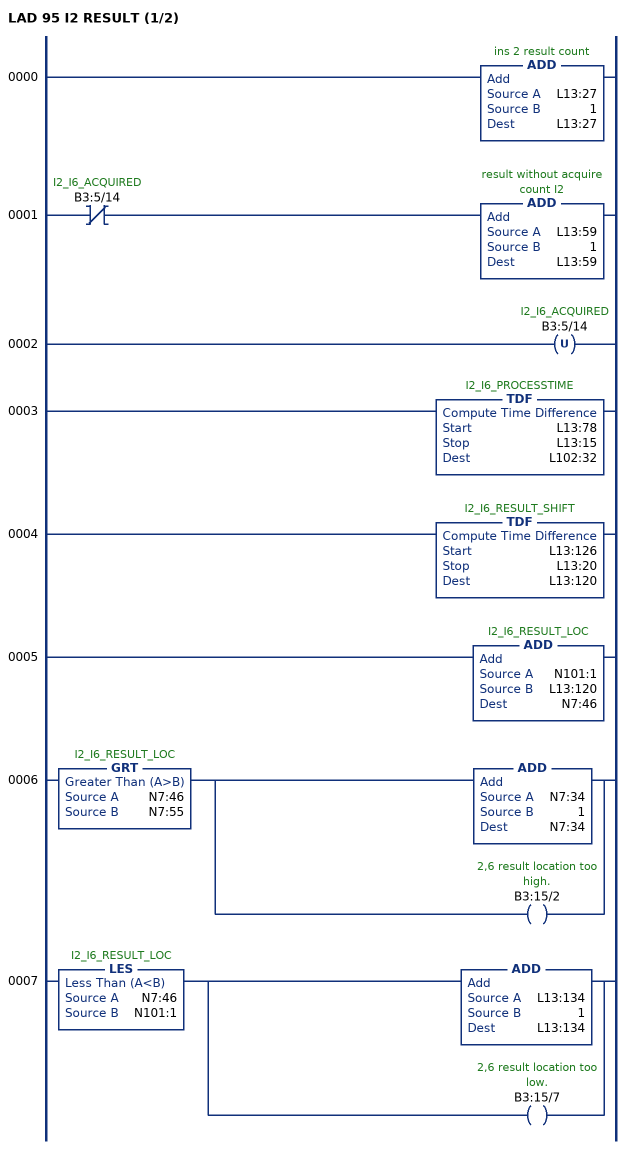
% Rung: 0 %
SOR ADD L13:27 1 L13:27 EOR
%   L13:27  "ins 2 result count" %
% Rung: 1 %
SOR XIO B3:5/14 ADD L13:59 1 L13:59 EOR
%   B3:5/14  I2_I6_ACQUIRED %
%   L13:59  "result without acquire count I2" %
% Rung: 2 %
SOR OTU B3:5/14 EOR
%   B3:5/14  I2_I6_ACQUIRED %
% Rung: 3 %
SOR TDF L13:78 L13:15 L102:32 EOR
%   L13:78  I2_I6_TIMEOFACQ %
%   L13:15  THE_TIME %
%   L102:32  I2_I6_PROCESSTIME %
% Rung: 4 %
SOR TDF L13:126 L13:20 L13:120 EOR
%   L13:126  I2_I6_PROC_START_POS %
%   L13:20  BOT_POSITION %
%   L13:120  I2_I6_RESULT_SHIFT %
% Rung: 5 %
SOR ADD N101:1 L13:120 N7:46 EOR
%   N101:1  I2_TRIG_LOC %
%   L13:120  I2_I6_RESULT_SHIFT %
%   N7:46  I2_I6_RESULT_LOC %
% Rung: 6 %
SOR GRT N7:46 N7:55 BST ADD N7:34 1 N7:34 NXB OTE B3:15/2 BND EOR
%   N7:46  I2_I6_RESULT_LOC %
%   N7:55  I2_MAX_SHIFT %
%   B3:15/2  "2,6 result location too high." %
% Rung: 7 %
SOR LES N7:46 N101:1 BST ADD L13:134 1 L13:134 NXB OTE B3:15/7 BND EOR
%   N7:46  I2_I6_RESULT_LOC %
%   N101:1  I2_TRIG_LOC %
%   B3:15/7  "2,6 result location too low." %

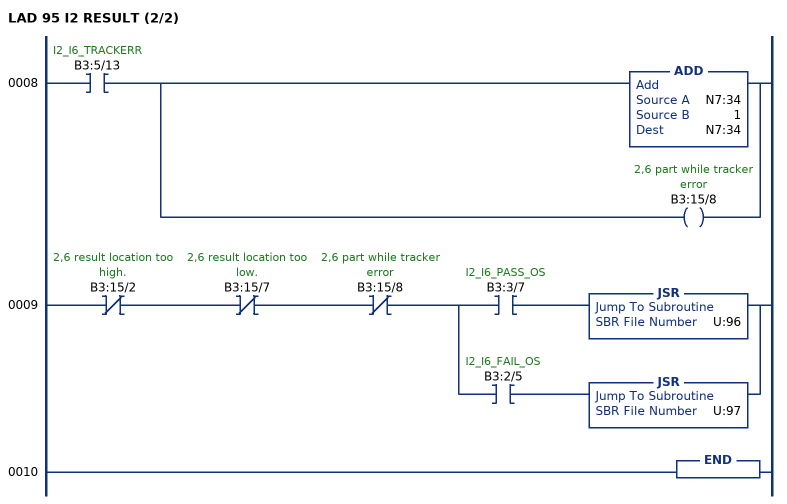
% Rung: 8 %
SOR XIC B3:5/13 BST ADD N7:34 1 N7:34 NXB OTE B3:15/8 BND EOR
%   B3:5/13  I2_I6_TRACKERR %
%   B3:15/8  "2,6 part while tracker error" %
% Rung: 9 %
SOR XIO B3:15/2 XIO B3:15/7 XIO B3:15/8 BST XIC B3:3/7 JSR U:96 NXB XIC B3:2/5 JSR U:97 BND EOR
%   B3:15/2  "2,6 result location too high." %
%   B3:15/7  "2,6 result location too low." %
%   B3:15/8  "2,6 part while tracker error" %
%   B3:3/7  I2_I6_PASS_OS %
%   B3:2/5  I2_I6_FAIL_OS %
% Rung: 10 %
SOR END EOR

LADDER 96 "I2 PASS"
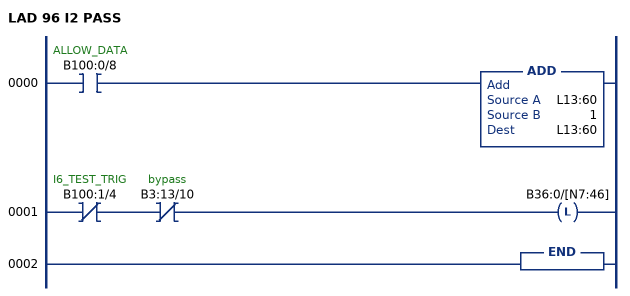
% Rung: 0 %
SOR XIC B100:0/8 ADD L13:60 1 L13:60 EOR
%   B100:0/8  ALLOW_DATA %
% Rung: 1 %
SOR XIO B100:1/4 XIO B3:13/10 OTL B36:0/[N7:46] EOR
%   B100:1/4  I6_TEST_TRIG %
%   B3:13/10  "bypass" %
%   B36:0  BOT_OK %
%   N7:46  I2_I6_RESULT_LOC %
% Rung: 2 %
SOR END EOR

LADDER 97 "I2 FAIL"
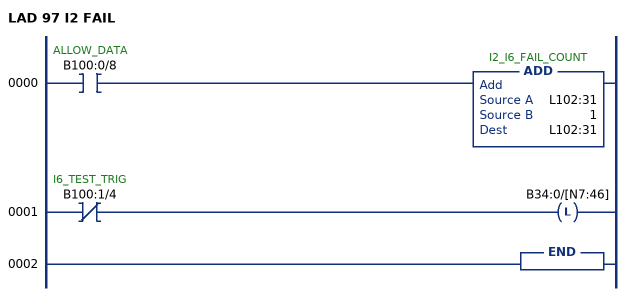
% Rung: 0 %
SOR XIC B100:0/8 ADD L102:31 1 L102:31 EOR
%   B100:0/8  ALLOW_DATA %
%   L102:31  I2_I6_FAIL_COUNT %
% Rung: 1 %
SOR XIO B100:1/4 OTL B34:0/[N7:46] EOR
%   B100:1/4  I6_TEST_TRIG %
%   B34:0  BOT_NG %
%   N7:46  I2_I6_RESULT_LOC %
% Rung: 2 %
SOR END EOR

LADDER 98 "I2 ACQ"
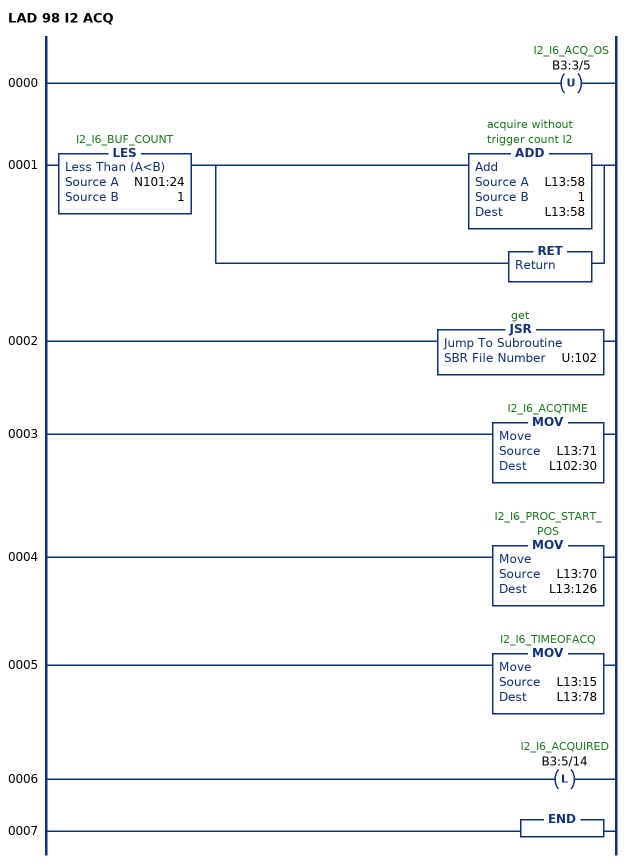
% Rung: 0 %
SOR OTU B3:3/5 EOR
%   B3:3/5  I2_I6_ACQ_OS %
% Rung: 1 %
SOR LES N101:24 1 BST ADD L13:58 1 L13:58 NXB RET BND EOR
%   N101:24  I2_I6_BUF_COUNT %
%   L13:58  "acquire without trigger count I2" %
% Rung: 2 %
SOR JSR U:102 EOR
%   U:102  "get" %
% Rung: 3 %
SOR MOV L13:71 L102:30 EOR
%   L13:71  I2_I6_TIME_SPAN %
%   L102:30  I2_I6_ACQTIME %
% Rung: 4 %
SOR MOV L13:70 L13:126 EOR
%   L13:70  I2_I6_PULLED_POS %
%   L13:126  I2_I6_PROC_START_POS %
% Rung: 5 %
SOR MOV L13:15 L13:78 EOR
%   L13:15  THE_TIME %
%   L13:78  I2_I6_TIMEOFACQ %
% Rung: 6 %
SOR OTL B3:5/14 EOR
%   B3:5/14  I2_I6_ACQUIRED %
% Rung: 7 %
SOR END EOR

LADDER 99 "I2 TESTER"
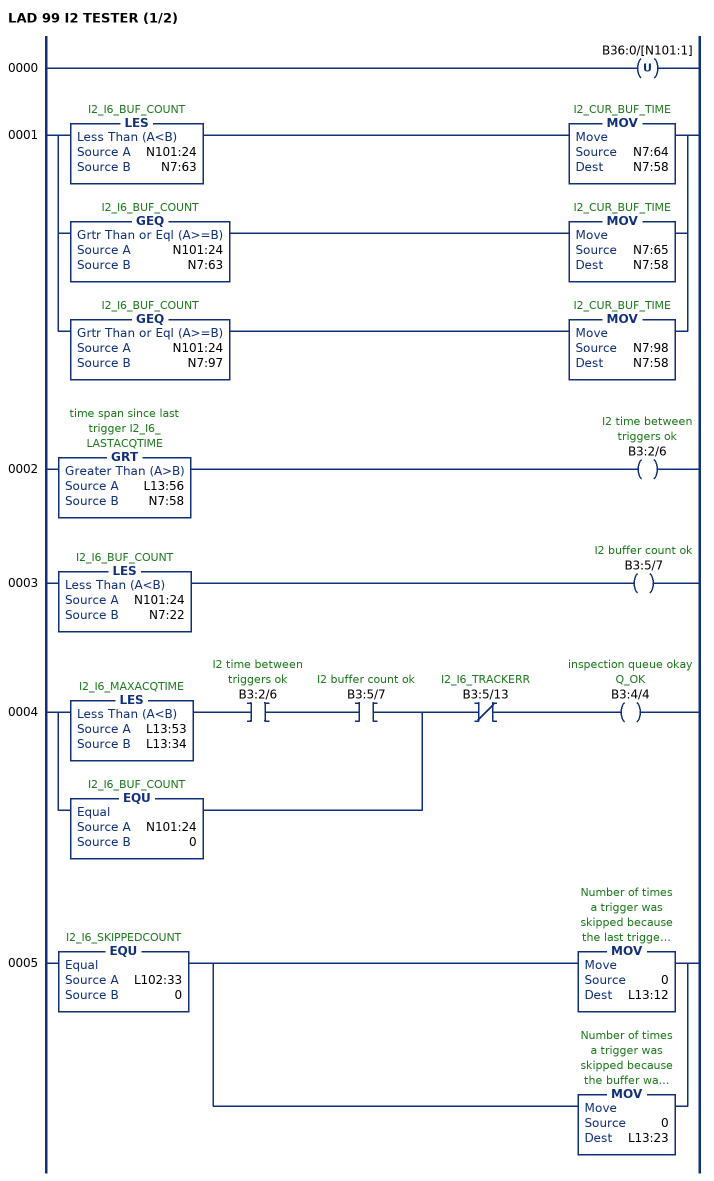
% Rung: 0 %
SOR OTU B36:0/[N101:1] EOR
%   B36:0  BOT_OK %
%   N101:1  I2_TRIG_LOC %
% Rung: 1 %
SOR BST LES N101:24 N7:63 MOV N7:64 N7:58 NXB GEQ N101:24 N7:63 MOV N7:65 N7:58 NXB GEQ N101:24 N7:97 MOV N7:98 N7:58 BND EOR
%   N101:24  I2_I6_BUF_COUNT %
%   N7:64  I2_CAM_BUF_TIME %
%   N7:58  I2_CUR_BUF_TIME %
%   N7:65  I2_PC_BUF_TIME %
% Rung: 2 %
SOR GRT L13:56 N7:58 OTE B3:2/6 EOR
%   L13:56  I2_I6_LASTACQTIME  "time span since last trigger" %
%   N7:58  I2_CUR_BUF_TIME %
%   B3:2/6  "I2 time between triggers ok" %
% Rung: 3 %
SOR LES N101:24 N7:22 OTE B3:5/7 EOR
%   N101:24  I2_I6_BUF_COUNT %
%   N7:22  MAX_BUF_ALL  "max buffer count alowed before bypass" %
%   B3:5/7  "I2 buffer count ok" %
% Rung: 4 %
SOR BST LES L13:53 L13:34 XIC B3:2/6 XIC B3:5/7 NXB EQU N101:24 0 BND XIO B3:5/13 OTE B3:4/4 EOR
%   L13:53  I2_I6_MAXACQTIME %
%   L13:34  MAX_ACQ_ALL  "absolute max acquire time before bypass trigger" %
%   B3:2/6  "I2 time between triggers ok" %
%   B3:5/7  "I2 buffer count ok" %
%   N101:24  I2_I6_BUF_COUNT %
%   B3:5/13  I2_I6_TRACKERR %
%   B3:4/4  Q_OK  "inspection queue okay" %
% Rung: 5 %
SOR EQU L102:33 0 BST MOV 0 L13:12 NXB MOV 0 L13:23 BND EOR
%   L102:33  I2_I6_SKIPPEDCOUNT %
%   L13:12  I2_FAST_TRIG_COUNT  "Number of times a trigger was skipped because the last trigger was too recent." %
%   L13:23  I2_BUF_FILL_COUNT  "Number of times a trigger was skipped because the buffer was full." %

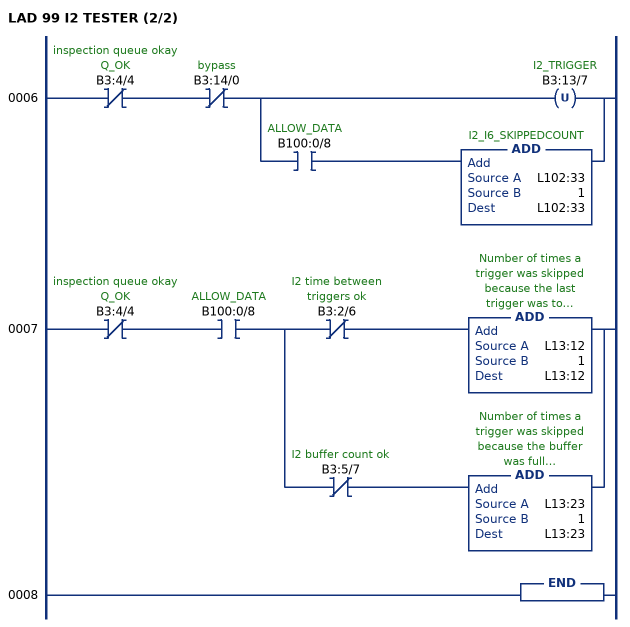
% Rung: 6 %
SOR XIO B3:4/4 XIO B3:14/0 BST OTU B3:13/7 NXB XIC B100:0/8 ADD L102:33 1 L102:33 BND EOR
%   B3:4/4  Q_OK  "inspection queue okay" %
%   B3:14/0  "bypass" %
%   B3:13/7  I2_TRIGGER %
%   B100:0/8  ALLOW_DATA %
%   L102:33  I2_I6_SKIPPEDCOUNT %
% Rung: 7 %
SOR XIO B3:4/4 XIC B100:0/8 BST XIO B3:2/6 ADD L13:12 1 L13:12 NXB XIO B3:5/7 ADD L13:23 1 L13:23 BND EOR
%   B3:4/4  Q_OK  "inspection queue okay" %
%   B100:0/8  ALLOW_DATA %
%   B3:2/6  "I2 time between triggers ok" %
%   L13:12  I2_FAST_TRIG_COUNT  "Number of times a trigger was skipped because the last trigger was too recent." %
%   B3:5/7  "I2 buffer count ok" %
%   L13:23  I2_BUF_FILL_COUNT  "Number of times a trigger was skipped because the buffer was full." %
% Rung: 8 %
SOR END EOR

LADDER 100 "I2 TRIG"
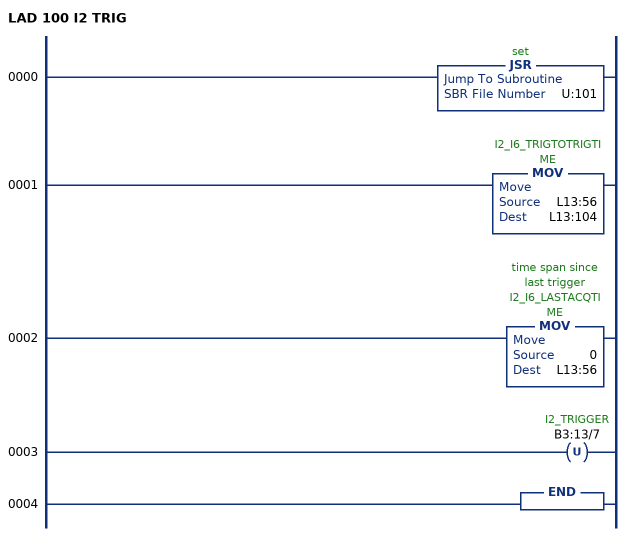
% Rung: 0 %
SOR JSR U:101 EOR
%   U:101  "set" %
% Rung: 1 %
SOR MOV L13:56 L13:104 EOR
%   L13:56  I2_I6_LASTACQTIME  "time span since last trigger" %
%   L13:104  I2_I6_TRIGTOTRIGTIME %
% Rung: 2 %
SOR MOV 0 L13:56 EOR
%   L13:56  I2_I6_LASTACQTIME  "time span since last trigger" %
% Rung: 3 %
SOR OTU B3:13/7 EOR
%   B3:13/7  I2_TRIGGER %
% Rung: 4 %
SOR END EOR

LADDER 101 "I2 FIFOSET"
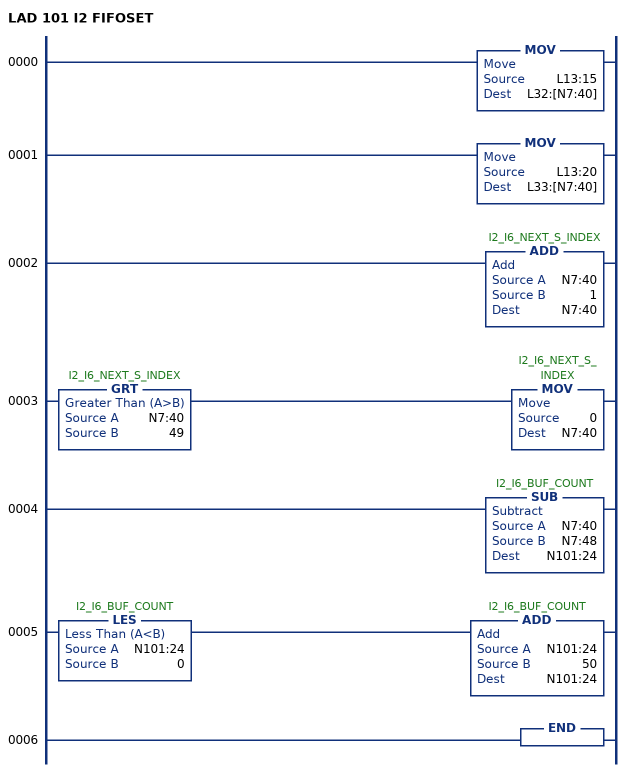
% Rung: 0 %
SOR MOV L13:15 L32:[N7:40] EOR
%   L13:15  THE_TIME %
%   N7:40  I2_I6_NEXT_S_INDEX %
% Rung: 1 %
SOR MOV L13:20 L33:[N7:40] EOR
%   L13:20  BOT_POSITION %
%   N7:40  I2_I6_NEXT_S_INDEX %
% Rung: 2 %
SOR ADD N7:40 1 N7:40 EOR
%   N7:40  I2_I6_NEXT_S_INDEX %
% Rung: 3 %
SOR GRT N7:40 49 MOV 0 N7:40 EOR
%   N7:40  I2_I6_NEXT_S_INDEX %
% Rung: 4 %
SOR SUB N7:40 N7:48 N101:24 EOR
%   N7:40  I2_I6_NEXT_S_INDEX %
%   N7:48  I2_I6_NEXT_G_INDEX %
%   N101:24  I2_I6_BUF_COUNT %
% Rung: 5 %
SOR LES N101:24 0 ADD N101:24 50 N101:24 EOR
%   N101:24  I2_I6_BUF_COUNT %
% Rung: 6 %
SOR END EOR

LADDER 102 "I2 FIFOGET"
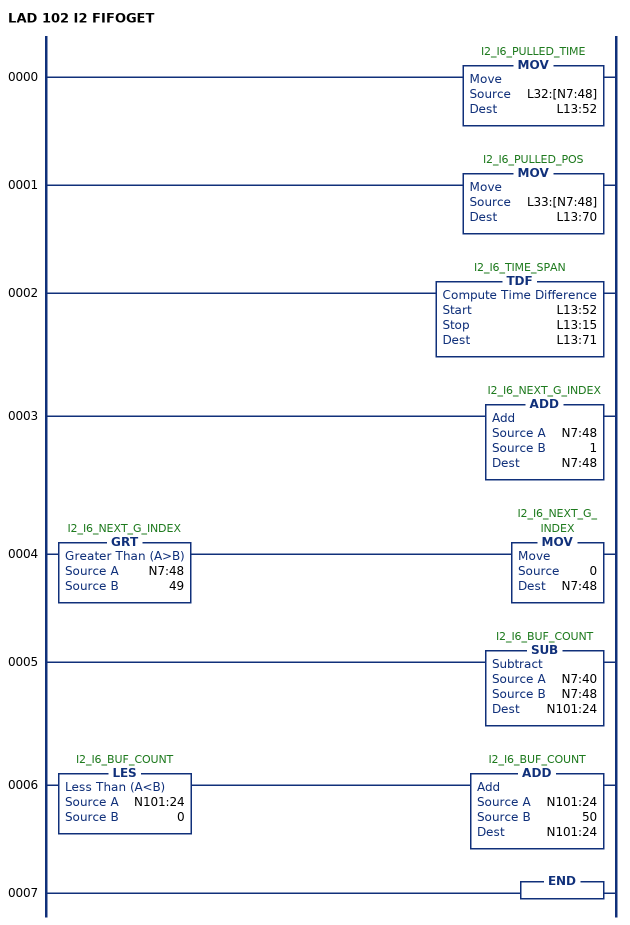
% Rung: 0 %
SOR MOV L32:[N7:48] L13:52 EOR
%   N7:48  I2_I6_NEXT_G_INDEX %
%   L13:52  I2_I6_PULLED_TIME %
% Rung: 1 %
SOR MOV L33:[N7:48] L13:70 EOR
%   N7:48  I2_I6_NEXT_G_INDEX %
%   L13:70  I2_I6_PULLED_POS %
% Rung: 2 %
SOR TDF L13:52 L13:15 L13:71 EOR
%   L13:52  I2_I6_PULLED_TIME %
%   L13:15  THE_TIME %
%   L13:71  I2_I6_TIME_SPAN %
% Rung: 3 %
SOR ADD N7:48 1 N7:48 EOR
%   N7:48  I2_I6_NEXT_G_INDEX %
% Rung: 4 %
SOR GRT N7:48 49 MOV 0 N7:48 EOR
%   N7:48  I2_I6_NEXT_G_INDEX %
% Rung: 5 %
SOR SUB N7:40 N7:48 N101:24 EOR
%   N7:40  I2_I6_NEXT_S_INDEX %
%   N7:48  I2_I6_NEXT_G_INDEX %
%   N101:24  I2_I6_BUF_COUNT %
% Rung: 6 %
SOR LES N101:24 0 ADD N101:24 50 N101:24 EOR
%   N101:24  I2_I6_BUF_COUNT %
% Rung: 7 %
SOR END EOR

LADDER 103 "I2 DATA"
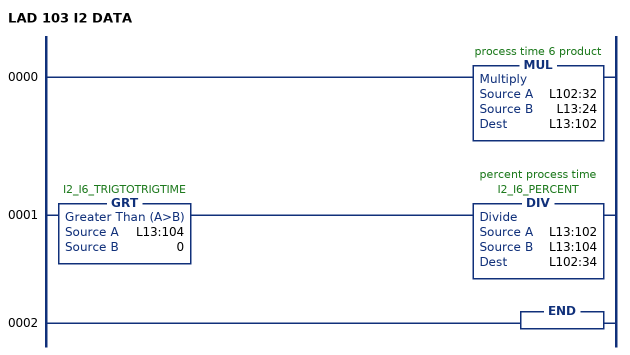
% Rung: 0 %
SOR MUL L102:32 L13:24 L13:102 EOR
%   L102:32  I2_I6_PROCESSTIME %
%   L13:24  "multiplyer to make devision come out to a percentage" %
%   L13:102  "process time 6 product" %
% Rung: 1 %
SOR GRT L13:104 0 DIV L13:102 L13:104 L102:34 EOR
%   L13:104  I2_I6_TRIGTOTRIGTIME %
%   L13:102  "process time 6 product" %
%   L102:34  I2_I6_PERCENT  "percent process time" %
% Rung: 2 %
SOR END EOR

LADDER 104 "I2 FAULT"
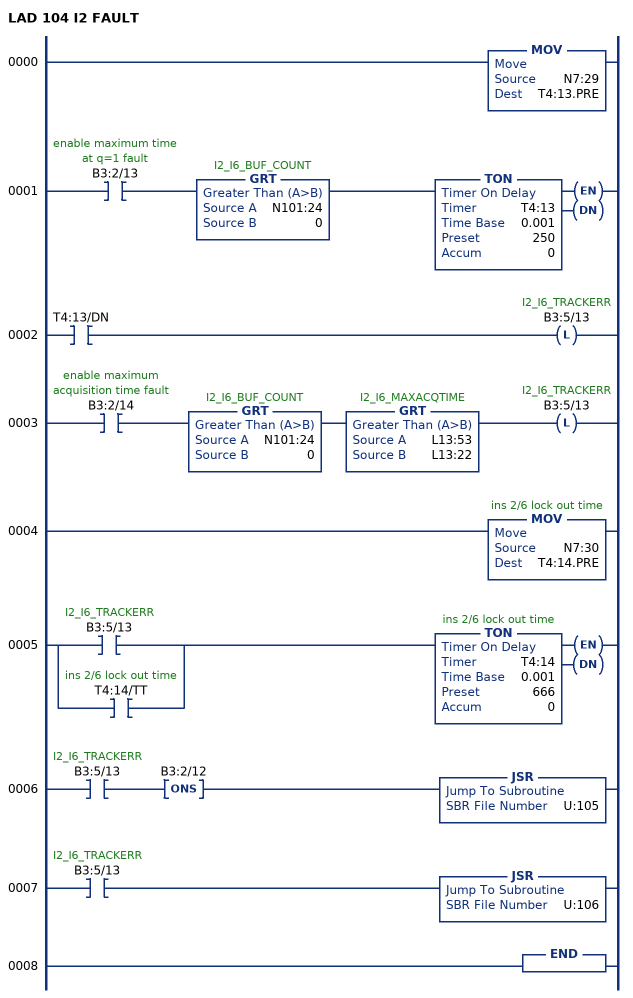
% Rung: 0 %
SOR MOV N7:29 T4:13.PRE EOR
%   N7:29  "max allowed ms time for q to be above 1 if safe fault is used" %
% Rung: 1 %
SOR XIC B3:2/13 GRT N101:24 0 TON T4:13 0.001 250 0 EOR
%   B3:2/13  "enable maximum time at q=1 fault" %
%   N101:24  I2_I6_BUF_COUNT %
% Rung: 2 %
SOR XIC T4:13/DN OTL B3:5/13 EOR
%   B3:5/13  I2_I6_TRACKERR %
% Rung: 3 %
SOR XIC B3:2/14 GRT N101:24 0 GRT L13:53 L13:22 OTL B3:5/13 EOR
%   B3:2/14  "enable maximum acquisition time fault" %
%   N101:24  I2_I6_BUF_COUNT %
%   L13:53  I2_I6_MAXACQTIME %
%   L13:22  "maximum of the longest acquire time allowed if maximum acquire time fault is enabled" %
%   B3:5/13  I2_I6_TRACKERR %
% Rung: 4 %
SOR MOV N7:30 T4:14.PRE EOR
%   N7:30  "ms time setting to lock out inspection to give all pending images a chance to clear" %
%   T4:14  "ins 2/6 lock out time" %
% Rung: 5 %
SOR BST XIC B3:5/13 NXB XIC T4:14/TT BND TON T4:14 0.001 666 0 EOR
%   B3:5/13  I2_I6_TRACKERR %
%   T4:14  "ins 2/6 lock out time" %
% Rung: 6 %
SOR XIC B3:5/13 ONS B3:2/12 JSR U:105 EOR
%   B3:5/13  I2_I6_TRACKERR %
% Rung: 7 %
SOR XIC B3:5/13 JSR U:106 EOR
%   B3:5/13  I2_I6_TRACKERR %
% Rung: 8 %
SOR END EOR

LADDER 105 "I2 FIX1"
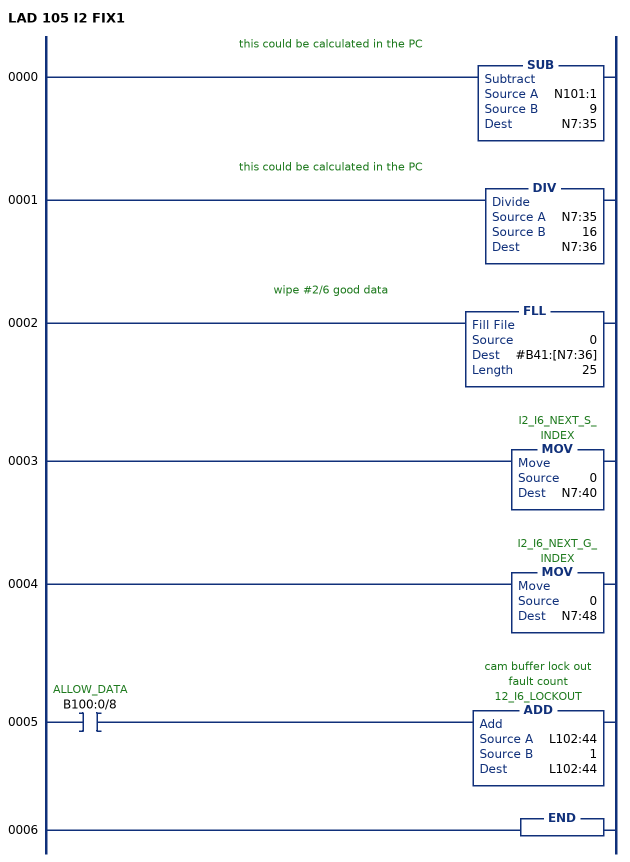
% Rung: 0 %
% this could be calculated in the PC %
SOR SUB N101:1 9 N7:35 EOR
%   N101:1  I2_TRIG_LOC %
% Rung: 1 %
% this could be calculated in the PC %
SOR DIV N7:35 16 N7:36 EOR
% Rung: 2 %
% wipe #2/6 good data %
SOR FLL 0 #B41:[N7:36] 25 EOR
% Rung: 3 %
SOR MOV 0 N7:40 EOR
%   N7:40  I2_I6_NEXT_S_INDEX %
% Rung: 4 %
SOR MOV 0 N7:48 EOR
%   N7:48  I2_I6_NEXT_G_INDEX %
% Rung: 5 %
SOR XIC B100:0/8 ADD L102:44 1 L102:44 EOR
%   B100:0/8  ALLOW_DATA %
%   L102:44  12_I6_LOCKOUT  "cam buffer lock out fault count" %
% Rung: 6 %
SOR END EOR

LADDER 106 "I2 FIX2"
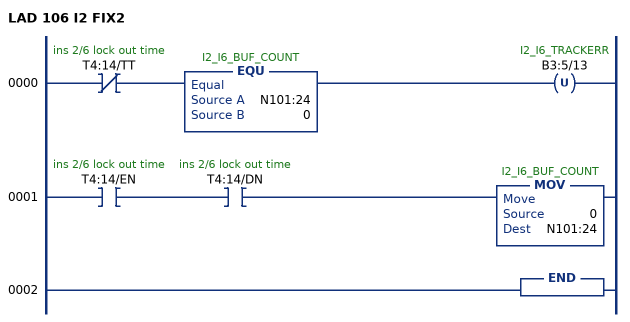
% Rung: 0 %
SOR XIO T4:14/TT EQU N101:24 0 OTU B3:5/13 EOR
%   T4:14  "ins 2/6 lock out time" %
%   N101:24  I2_I6_BUF_COUNT %
%   B3:5/13  I2_I6_TRACKERR %
% Rung: 1 %
SOR XIC T4:14/EN XIC T4:14/DN MOV 0 N101:24 EOR
%   T4:14  "ins 2/6 lock out time" %
%   N101:24  I2_I6_BUF_COUNT %
% Rung: 2 %
SOR END EOR

LADDER 135 "XFER"
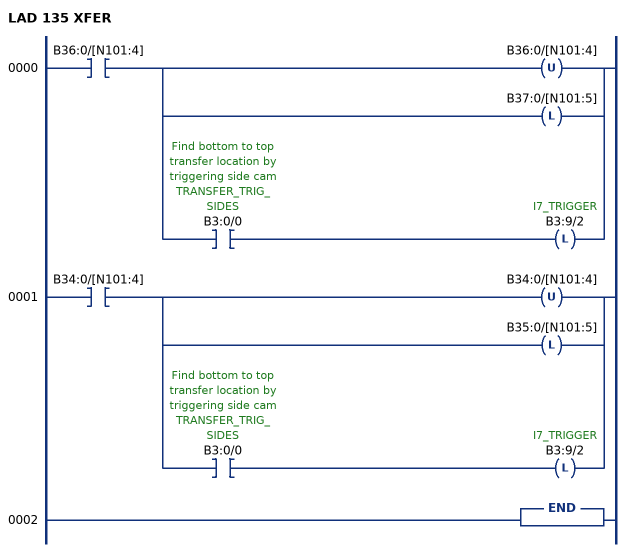
% Rung: 0 %
SOR XIC B36:0/[N101:4] BST OTU B36:0/[N101:4] NXB OTL B37:0/[N101:5] NXB XIC B3:0/0 OTL B3:9/2 BND EOR
%   B36:0  BOT_OK %
%   N101:4  XFER_OUT_LOC %
%   B37:0  TOP_OK_1 %
%   N101:5  XFER_IN_LOC %
%   B3:0/0  TRANSFER_TRIG_SIDES  "Find bottom to top transfer location by triggering side cam" %
%   B3:9/2  I7_TRIGGER %
% Rung: 1 %
SOR XIC B34:0/[N101:4] BST OTU B34:0/[N101:4] NXB OTL B35:0/[N101:5] NXB XIC B3:0/0 OTL B3:9/2 BND EOR
%   B34:0  BOT_NG %
%   N101:4  XFER_OUT_LOC %
%   B35:0  TOP_NG %
%   N101:5  XFER_IN_LOC %
%   B3:0/0  TRANSFER_TRIG_SIDES  "Find bottom to top transfer location by triggering side cam" %
%   B3:9/2  I7_TRIGGER %
% Rung: 2 %
SOR END EOR

LADDER 137 "TOPOPTIC"
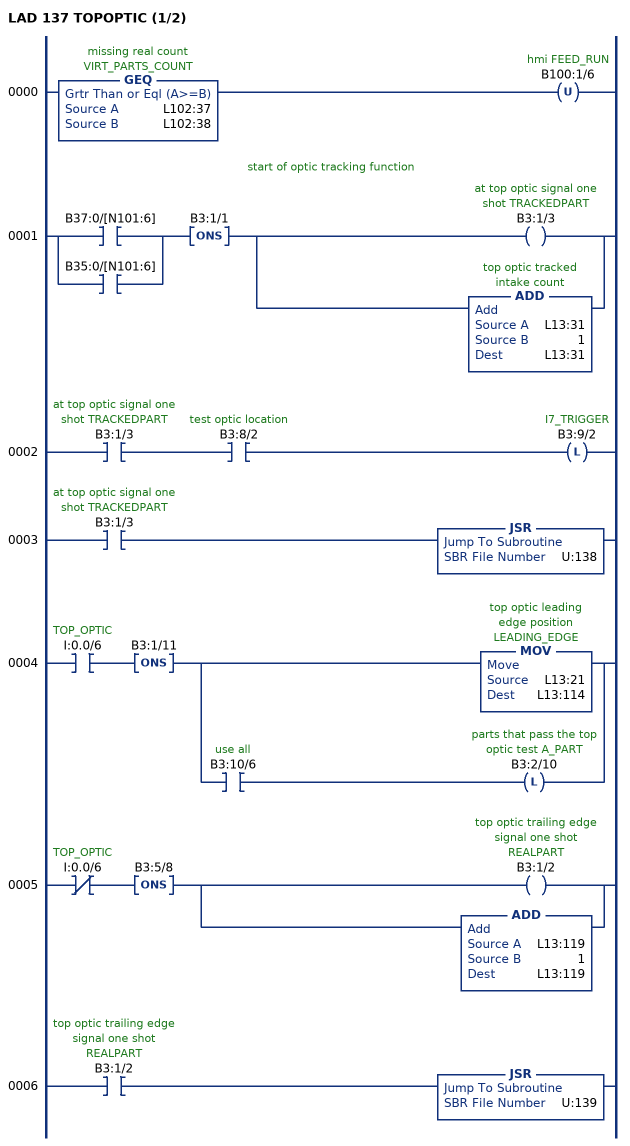
% Rung: 0 %
SOR GEQ L102:37 L102:38 OTU B100:1/6 EOR
%   L102:37  VIRT_PARTS_COUNT  "missing real count" %
%   L102:38  FELL_PARTS_LIMIT %
%   B100:1/6  FEED_RUN  "hmi" %
% Rung: 1 %
% start of optic tracking function %
SOR BST XIC B37:0/[N101:6] NXB XIC B35:0/[N101:6] BND ONS B3:1/1 BST OTE B3:1/3 NXB ADD L13:31 1 L13:31 BND EOR
%   B37:0  TOP_OK_1 %
%   N101:6  TOP_OPTIC_LOC %
%   B35:0  TOP_NG %
%   B3:1/3  TRACKEDPART  "at top optic signal one shot" %
%   L13:31  "top optic tracked intake count" %
% Rung: 2 %
SOR XIC B3:1/3 XIC B3:8/2 OTL B3:9/2 EOR
%   B3:1/3  TRACKEDPART  "at top optic signal one shot" %
%   B3:8/2  "test optic location" %
%   B3:9/2  I7_TRIGGER %
% Rung: 3 %
SOR XIC B3:1/3 JSR U:138 EOR
%   B3:1/3  TRACKEDPART  "at top optic signal one shot" %
% Rung: 4 %
SOR XIC I:0.0/6 ONS B3:1/11 BST MOV L13:21 L13:114 NXB XIC B3:10/6 OTL B3:2/10 BND EOR
%   I:0.0/6  TOP_OPTIC %
%   L13:21  TOP_POSITION %
%   L13:114  LEADING_EDGE  "top optic leading edge position" %
%   B3:10/6  "use all" %
%   B3:2/10  A_PART  "parts that pass the top optic test" %
% Rung: 5 %
SOR XIO I:0.0/6 ONS B3:5/8 BST OTE B3:1/2 NXB ADD L13:119 1 L13:119 BND EOR
%   I:0.0/6  TOP_OPTIC %
%   B3:1/2  REALPART  "top optic trailing edge signal one shot" %
% Rung: 6 %
SOR XIC B3:1/2 JSR U:139 EOR
%   B3:1/2  REALPART  "top optic trailing edge signal one shot" %

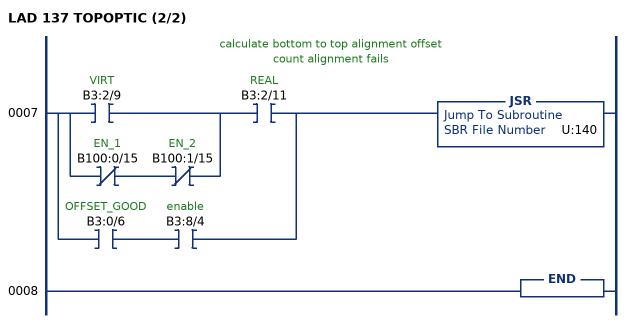
% Rung: 7 %
% calculate bottom to top alignment offset
% count alignment fails %
SOR BST BST XIC B3:2/9 NXB XIO B100:0/15 XIO B100:1/15 BND XIC B3:2/11 NXB XIC B3:0/6 XIC B3:8/4 BND JSR U:140 EOR
%   B3:2/9  VIRT %
%   B100:0/15  EN_1 %
%   B100:1/15  EN_2 %
%   B3:2/11  REAL %
%   B3:0/6  OFFSET_GOOD %
%   B3:8/4  "enable" %
% Rung: 8 %
SOR END EOR

LADDER 138 "TOPOPVERT"
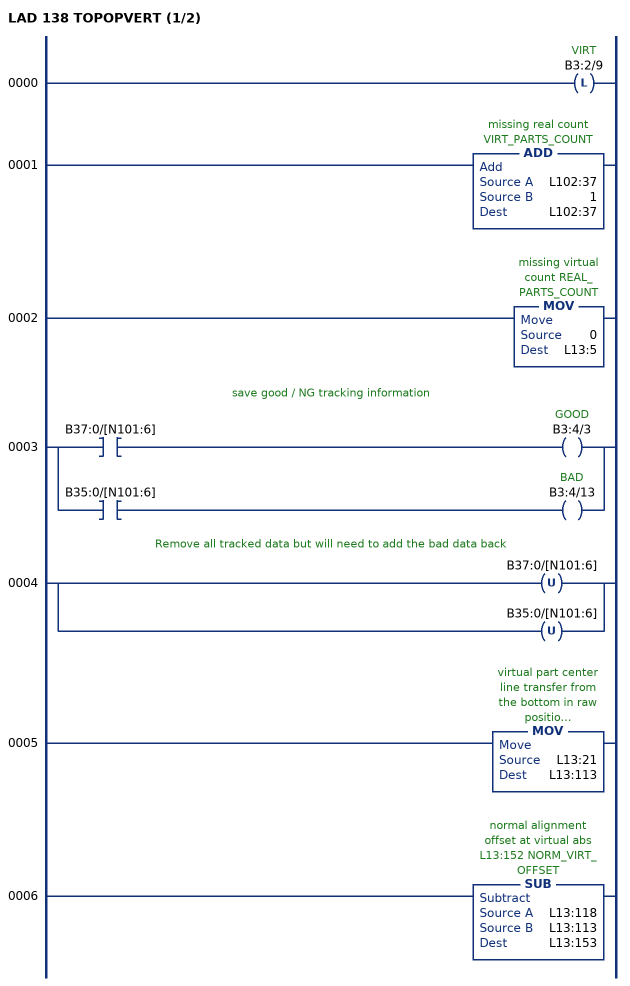
% Rung: 0 %
SOR OTL B3:2/9 EOR
%   B3:2/9  VIRT %
% Rung: 1 %
SOR ADD L102:37 1 L102:37 EOR
%   L102:37  VIRT_PARTS_COUNT  "missing real count" %
% Rung: 2 %
SOR MOV 0 L13:5 EOR
%   L13:5  REAL_PARTS_COUNT  "missing virtual count" %
% Rung: 3 %
% save good / NG tracking information %
SOR BST XIC B37:0/[N101:6] OTE B3:4/3 NXB XIC B35:0/[N101:6] OTE B3:4/13 BND EOR
%   B37:0  TOP_OK_1 %
%   N101:6  TOP_OPTIC_LOC %
%   B3:4/3  GOOD %
%   B35:0  TOP_NG %
%   B3:4/13  BAD %
% Rung: 4 %
% Remove all tracked data but will need to add the bad data back %
SOR BST OTU B37:0/[N101:6] NXB OTU B35:0/[N101:6] BND EOR
%   B37:0  TOP_OK_1 %
%   N101:6  TOP_OPTIC_LOC %
%   B35:0  TOP_NG %
% Rung: 5 %
SOR MOV L13:21 L13:113 EOR
%   L13:21  TOP_POSITION %
%   L13:113  VIRT_CL_POSITION  "virtual part center line transfer from the bottom in raw position" %
% Rung: 6 %
SOR SUB L13:118 L13:113 L13:153 EOR
%   L13:118  REAL_CL_POSITION  "real part center line in raw position" %
%   L13:113  VIRT_CL_POSITION  "virtual part center line transfer from the bottom in raw position" %
%   L13:153  NORM_VIRT_OFFSET  "normal alignment offset at virtual abs L13:152" %

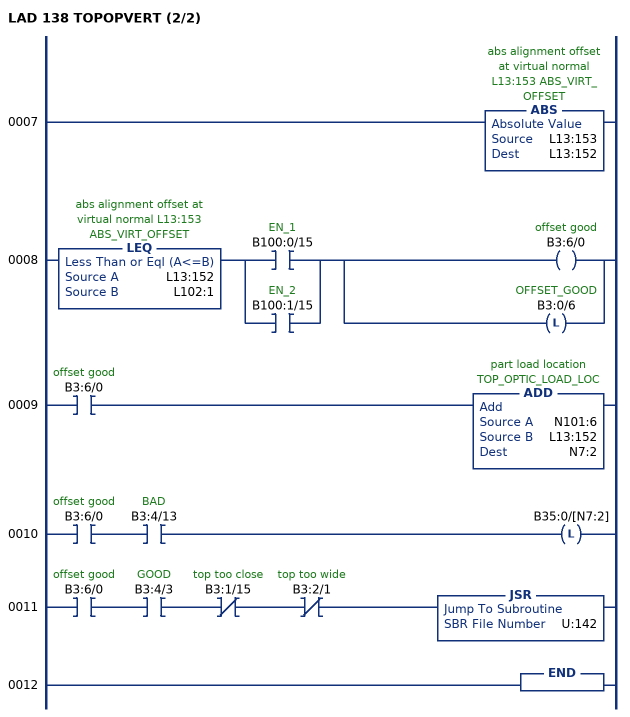
% Rung: 7 %
SOR ABS L13:153 L13:152 EOR
%   L13:153  NORM_VIRT_OFFSET  "normal alignment offset at virtual abs L13:152" %
%   L13:152  ABS_VIRT_OFFSET  "abs alignment offset at virtual normal L13:153" %
% Rung: 8 %
SOR LEQ L13:152 L102:1 BST XIC B100:0/15 NXB XIC B100:1/15 BND BST OTE B3:6/0 NXB OTL B3:0/6 BND EOR
%   L13:152  ABS_VIRT_OFFSET  "abs alignment offset at virtual normal L13:153" %
%   L102:1  MAX_OFFSET  "transition zone width" %
%   B100:0/15  EN_1 %
%   B100:1/15  EN_2 %
%   B3:6/0  "offset good" %
%   B3:0/6  OFFSET_GOOD %
% Rung: 9 %
SOR XIC B3:6/0 ADD N101:6 L13:152 N7:2 EOR
%   B3:6/0  "offset good" %
%   N101:6  TOP_OPTIC_LOC %
%   L13:152  ABS_VIRT_OFFSET  "abs alignment offset at virtual normal L13:153" %
%   N7:2  TOP_OPTIC_LOAD_LOC  "part load location" %
% Rung: 10 %
SOR XIC B3:6/0 XIC B3:4/13 OTL B35:0/[N7:2] EOR
%   B3:6/0  "offset good" %
%   B3:4/13  BAD %
%   B35:0  TOP_NG %
%   N7:2  TOP_OPTIC_LOAD_LOC  "part load location" %
% Rung: 11 %
SOR XIC B3:6/0 XIC B3:4/3 XIO B3:1/15 XIO B3:2/1 JSR U:142 EOR
%   B3:6/0  "offset good" %
%   B3:4/3  GOOD %
%   B3:1/15  "top too close" %
%   B3:2/1  "top too wide" %
% Rung: 12 %
SOR END EOR

LADDER 139 "TOPOPREAL"
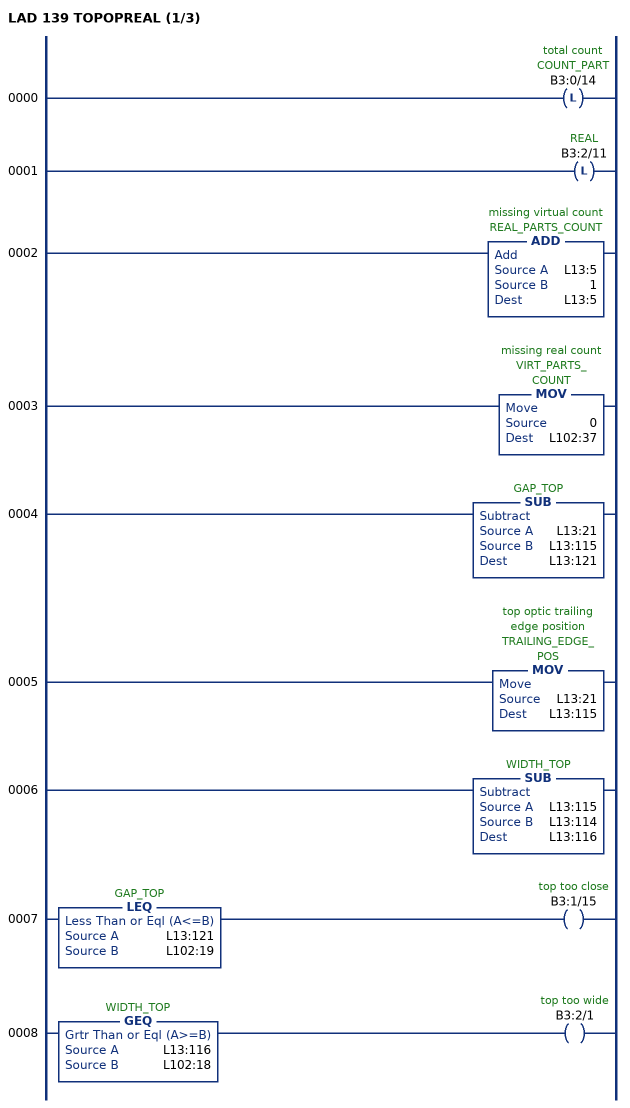
% Rung: 0 %
SOR OTL B3:0/14 EOR
%   B3:0/14  COUNT_PART  "total count" %
% Rung: 1 %
SOR OTL B3:2/11 EOR
%   B3:2/11  REAL %
% Rung: 2 %
SOR ADD L13:5 1 L13:5 EOR
%   L13:5  REAL_PARTS_COUNT  "missing virtual count" %
% Rung: 3 %
SOR MOV 0 L102:37 EOR
%   L102:37  VIRT_PARTS_COUNT  "missing real count" %
% Rung: 4 %
SOR SUB L13:21 L13:115 L13:121 EOR
%   L13:21  TOP_POSITION %
%   L13:115  TRAILING_EDGE_POS  "top optic trailing edge position" %
%   L13:121  GAP_TOP %
% Rung: 5 %
SOR MOV L13:21 L13:115 EOR
%   L13:21  TOP_POSITION %
%   L13:115  TRAILING_EDGE_POS  "top optic trailing edge position" %
% Rung: 6 %
SOR SUB L13:115 L13:114 L13:116 EOR
%   L13:115  TRAILING_EDGE_POS  "top optic trailing edge position" %
%   L13:114  LEADING_EDGE  "top optic leading edge position" %
%   L13:116  WIDTH_TOP %
% Rung: 7 %
SOR LEQ L13:121 L102:19 OTE B3:1/15 EOR
%   L13:121  GAP_TOP %
%   L102:19  MIN_GAP_TOP %
%   B3:1/15  "top too close" %
% Rung: 8 %
SOR GEQ L13:116 L102:18 OTE B3:2/1 EOR
%   L13:116  WIDTH_TOP %
%   L102:18  MAX_WIDTH_TOP %
%   B3:2/1  "top too wide" %

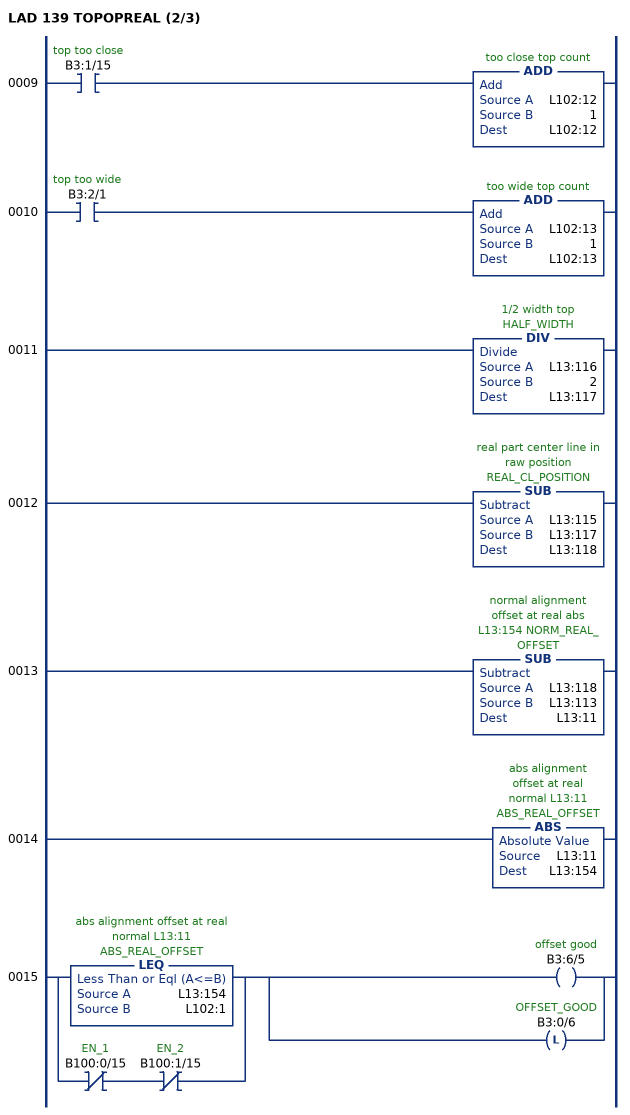
% Rung: 9 %
SOR XIC B3:1/15 ADD L102:12 1 L102:12 EOR
%   B3:1/15  "top too close" %
%   L102:12  "too close top count" %
% Rung: 10 %
SOR XIC B3:2/1 ADD L102:13 1 L102:13 EOR
%   B3:2/1  "top too wide" %
%   L102:13  "too wide top count" %
% Rung: 11 %
SOR DIV L13:116 2 L13:117 EOR
%   L13:116  WIDTH_TOP %
%   L13:117  HALF_WIDTH  "1/2 width top" %
% Rung: 12 %
SOR SUB L13:115 L13:117 L13:118 EOR
%   L13:115  TRAILING_EDGE_POS  "top optic trailing edge position" %
%   L13:117  HALF_WIDTH  "1/2 width top" %
%   L13:118  REAL_CL_POSITION  "real part center line in raw position" %
% Rung: 13 %
SOR SUB L13:118 L13:113 L13:11 EOR
%   L13:118  REAL_CL_POSITION  "real part center line in raw position" %
%   L13:113  VIRT_CL_POSITION  "virtual part center line transfer from the bottom in raw position" %
%   L13:11  NORM_REAL_OFFSET  "normal alignment offset at real abs L13:154" %
% Rung: 14 %
SOR ABS L13:11 L13:154 EOR
%   L13:11  NORM_REAL_OFFSET  "normal alignment offset at real abs L13:154" %
%   L13:154  ABS_REAL_OFFSET  "abs alignment offset at real normal L13:11" %
% Rung: 15 %
SOR BST LEQ L13:154 L102:1 NXB XIO B100:0/15 XIO B100:1/15 BND BST OTE B3:6/5 NXB OTL B3:0/6 BND EOR
%   L13:154  ABS_REAL_OFFSET  "abs alignment offset at real normal L13:11" %
%   L102:1  MAX_OFFSET  "transition zone width" %
%   B100:0/15  EN_1 %
%   B100:1/15  EN_2 %
%   B3:6/5  "offset good" %
%   B3:0/6  OFFSET_GOOD %

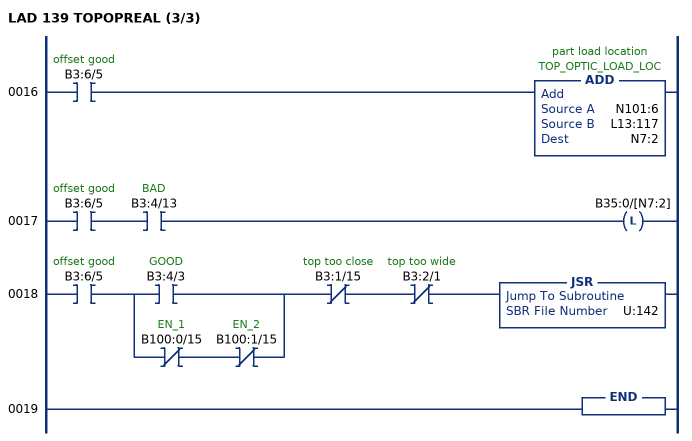
% Rung: 16 %
SOR XIC B3:6/5 ADD N101:6 L13:117 N7:2 EOR
%   B3:6/5  "offset good" %
%   N101:6  TOP_OPTIC_LOC %
%   L13:117  HALF_WIDTH  "1/2 width top" %
%   N7:2  TOP_OPTIC_LOAD_LOC  "part load location" %
% Rung: 17 %
SOR XIC B3:6/5 XIC B3:4/13 OTL B35:0/[N7:2] EOR
%   B3:6/5  "offset good" %
%   B3:4/13  BAD %
%   B35:0  TOP_NG %
%   N7:2  TOP_OPTIC_LOAD_LOC  "part load location" %
% Rung: 18 %
SOR XIC B3:6/5 BST XIC B3:4/3 NXB XIO B100:0/15 XIO B100:1/15 BND XIO B3:1/15 XIO B3:2/1 JSR U:142 EOR
%   B3:6/5  "offset good" %
%   B3:4/3  GOOD %
%   B100:0/15  EN_1 %
%   B100:1/15  EN_2 %
%   B3:1/15  "top too close" %
%   B3:2/1  "top too wide" %
% Rung: 19 %
SOR END EOR

LADDER 140 "CT ALIGNS"
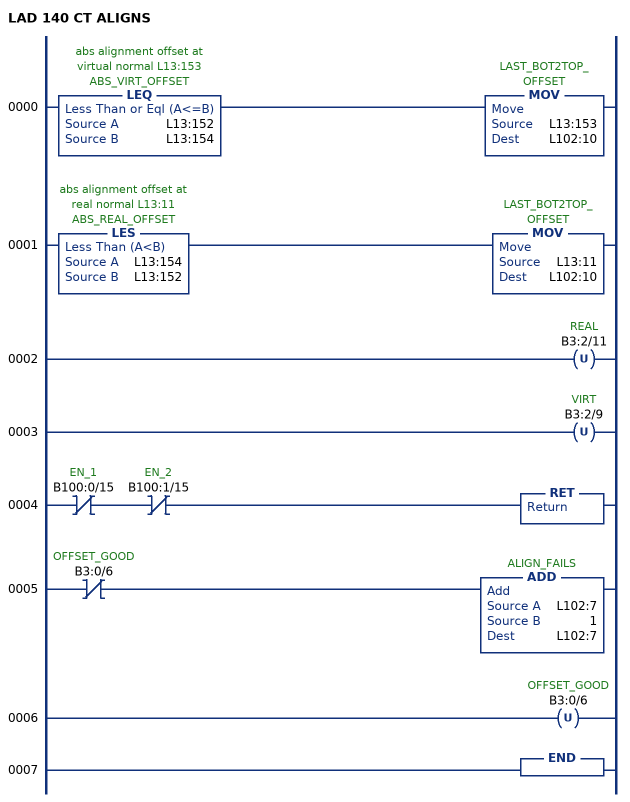
% Rung: 0 %
SOR LEQ L13:152 L13:154 MOV L13:153 L102:10 EOR
%   L13:152  ABS_VIRT_OFFSET  "abs alignment offset at virtual normal L13:153" %
%   L13:154  ABS_REAL_OFFSET  "abs alignment offset at real normal L13:11" %
%   L13:153  NORM_VIRT_OFFSET  "normal alignment offset at virtual abs L13:152" %
%   L102:10  LAST_BOT2TOP_OFFSET %
% Rung: 1 %
SOR LES L13:154 L13:152 MOV L13:11 L102:10 EOR
%   L13:154  ABS_REAL_OFFSET  "abs alignment offset at real normal L13:11" %
%   L13:152  ABS_VIRT_OFFSET  "abs alignment offset at virtual normal L13:153" %
%   L13:11  NORM_REAL_OFFSET  "normal alignment offset at real abs L13:154" %
%   L102:10  LAST_BOT2TOP_OFFSET %
% Rung: 2 %
SOR OTU B3:2/11 EOR
%   B3:2/11  REAL %
% Rung: 3 %
SOR OTU B3:2/9 EOR
%   B3:2/9  VIRT %
% Rung: 4 %
SOR XIO B100:0/15 XIO B100:1/15 RET EOR
%   B100:0/15  EN_1 %
%   B100:1/15  EN_2 %
% Rung: 5 %
SOR XIO B3:0/6 ADD L102:7 1 L102:7 EOR
%   B3:0/6  OFFSET_GOOD %
%   L102:7  ALIGN_FAILS %
% Rung: 6 %
SOR OTU B3:0/6 EOR
%   B3:0/6  OFFSET_GOOD %
% Rung: 7 %
SOR END EOR

LADDER 142 "SET GOOD"
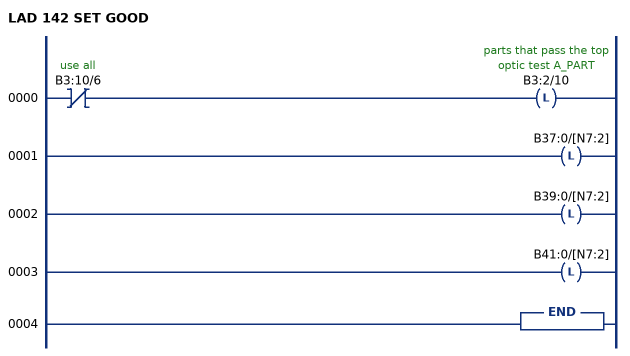
% Rung: 0 %
SOR XIO B3:10/6 OTL B3:2/10 EOR
%   B3:10/6  "use all" %
%   B3:2/10  A_PART  "parts that pass the top optic test" %
% Rung: 1 %
SOR OTL B37:0/[N7:2] EOR
%   B37:0  TOP_OK_1 %
%   N7:2  TOP_OPTIC_LOAD_LOC  "part load location" %
% Rung: 2 %
SOR OTL B39:0/[N7:2] EOR
%   B39:0  TOP_OK_2 %
%   N7:2  TOP_OPTIC_LOAD_LOC  "part load location" %
% Rung: 3 %
SOR OTL B41:0/[N7:2] EOR
%   B41:0  TOP_OK_3 %
%   N7:2  TOP_OPTIC_LOAD_LOC  "part load location" %
% Rung: 4 %
SOR END EOR

LADDER 148 "I5"
